{attribute 'GeneratedUsingTerminal: ATH2050-5501-0022'}
{attribute addProperty BoxType "ATH2050-5501-0022"}
{attribute addProperty Id "BinaryDataAT %I*ARRAY [0..55] OF BYTE0"}
{attribute addProperty CRC "957634129"}
{attribute addProperty Size "0"}
TYPE FB_Inputs_39145651 :
STRUCT
	{attribute addProperty Name "BinaryData"}
	BinaryData AT %I* : ARRAY [0..55] OF BYTE;
END_STRUCT
END_TYPE

(* stored: Version 1.2.0.0, ProductVersion 3.1.4024.9
   DUT FB_Inputs_39145651: Id {35aec4a3-7444-4e0e-a03d-6dd3dfbe90ca} *)
